TYPE StatusStructExtended :
STRUCT
	Enabled: BIT;
	Tripped : BIT;
	ShortCircuit : BIT;
	Overload : BIT;
	HWProtection : BIT;
	Overvoltage : BIT;
	Undervoltage : BIT;
	CurrentLevelWarning : BIT;
	
	CoolDownLock : BIT;
	DisabledBySwitch : BIT;
	DisabledByDI : BIT;
	DisabledByOutput : BIT;
	Diag : BIT;
	TxPDOState : BIT;
	InputCycleCount : BIT;
	InputCycleCount2 : BIT;
	
	StateDeviceSwitch : BIT;
	StateDigitalInput : BIT;
	Error : BIT;
	StateReset : BIT;
	StateSwitch : BIT;
	{attribute 'hide'}
	_hidden_bit_0: BIT;
	{attribute 'hide'}
	_hidden_bit_1: BIT;
	{attribute 'hide'}
	_hidden_bit_2: BIT;
	{attribute 'hide'}
	_hidden_byte_0: BYTE;
END_STRUCT
END_TYPE

(* stored: Version 1.1.0.1, ProductVersion 3.1.4024.5
   DUT StatusStructExtended: Id {2a641705-ab07-42d5-9d4f-08c804024823} *)
